INTERFACE itfAxis_Tc2_MC2

METHOD AbortTrigger : itfCommand
VAR_INPUT
END_VAR
END_METHOD

{attribute 'TcRpcEnable'}
METHOD AccelerationProfile 	: itfCommand
VAR_INPUT
	TimeScale				: REAL;
	AccelerationScale		: REAL;
	Offset					: REAL;
	BufferMode				: MC_BUFFER_MODE;
END_VAR
END_METHOD

{warning 'add property implementation'}
PROPERTY ActualPosition : REAL
GET
END_GET
END_PROPERTY

{warning 'add property implementation'}
PROPERTY ActualTorque : REAL
GET
END_GET
END_PROPERTY

{warning 'add property implementation'}
PROPERTY ActualVelocity : REAL
GET
END_GET
END_PROPERTY

{warning 'add property implementation'}
PROPERTY AxisWarning : BOOL
GET
END_GET
END_PROPERTY

{attribute 'TcRpcEnable'}
METHOD CombineAxes 			: itfSynchronizedAxisCommand
VAR_INPUT
	Master1					: itfAxis_Tc2_MC2;
	Master2					: itfAxis_Tc2_MC2;
	CombineMode				: MC_COMBINE_MODE;
	GearRatioNumeratorM1	: INT;
	GearRatioDenominatorM1	: INT;
	GearRatioNumeratorM2	: INT;
	GearRatioDenominatorM2	: INT;
	MasterValueSourceM1		: MC_SOURCE;
	MasterValueSourceM2		: MC_SOURCE;
	BufferMode				: MC_BUFFER_MODE;
END_VAR
END_METHOD

{warning 'add property implementation'}
PROPERTY CommunicationReady : BOOL
GET
END_GET
END_PROPERTY

{warning 'add property implementation'}
PROPERTY Direction : AXIS_DIRECTION
GET
END_GET
END_PROPERTY

PROPERTY Error : BOOL
GET
END_GET
END_PROPERTY

{warning 'add property implementation'}
PROPERTY ErrorId : WORD
GET
END_GET
END_PROPERTY

PROPERTY ErrorId_Udint_Status : UDINT
GET
END_GET
END_PROPERTY

PROPERTY Geared : BOOL
GET
END_GET
END_PROPERTY

{attribute 'TcRpcEnable'}
METHOD GearIn 			: itfSynchronizedAxisCommand
VAR_INPUT
//	Master				: itfAxis;
//	Master				: Tc2_MC2.AXIS_REF;
//	Slave				: Tc2_MC2.AXIS_REF;		
//	Ratio				: REAL;
//	MasterValueSource	: INT;
	RatioNumerator		: LREAL;
	RatioDenominator	: UINT;
	Acceleration		: REAL;
	Deceleration		: REAL;
	Jerk				: REAL;
	BufferMode			: MC_BUFFER_MODE;
//	BufferMode			: Tc2_MC2.MC_BufferMode;
//	Options             : Tc2_MC2.ST_GearInOptions;
END_VAR

VAR_IN_OUT 
	Slave				: Tc2_MC2.AXIS_REF;	
END_VAR
END_METHOD

{attribute 'TcRpcEnable'}
METHOD Halt 		: itfAxisCommand
VAR_INPUT
	Deceleration	: REAL;
	Jerk			: REAL;
	BufferMode		: MC_BUFFER_MODE;
END_VAR
END_METHOD

{attribute 'TcRpcEnable'}
METHOD HaltSuperimposed : itfAxisCommand
VAR_INPUT
	Deceleration		: REAL;
	Jerk				: REAL;
END_VAR
END_METHOD

{attribute 'TcRpcEnable'}
METHOD Home 		: itfAxisCommand
VAR_INPUT
	Position		: REAL;
	Velocity		: REAL;
	EndVelocity		: REAL;
	Acceleration	: REAL;
	Deceleration	: REAL;
	Jerk			: REAL;
	Direction		: MC_Direction;
	HomingMode		: INT;
	BufferMode		: MC_BUFFER_MODE;
END_VAR
END_METHOD

{warning 'add property implementation'}
PROPERTY HomeAbsSwitch : BOOL
GET
END_GET
END_PROPERTY


PROPERTY IsHomed : BOOL
GET
END_GET
END_PROPERTY

{attribute 'TcRpcEnable'}
METHOD Jog 			: itfAxisCommand
VAR_INPUT
    JogForward 		: BOOL;
    JogBackwards 	: BOOL;
    Mode     		: Tc2_MC2.E_JogMode;
    Position        : LREAL;
    Velocity        : LREAL;
    Acceleration 	: LREAL;
    Deceleration 	: LREAL;
    Jerk     		: LREAL;
END_VAR
END_METHOD

{warning 'add property implementation'}
PROPERTY LimitSwitchNegative : BOOL
GET
END_GET
END_PROPERTY

{warning 'add property implementation'}
PROPERTY LimitSwitchPositive : BOOL
GET
END_GET
END_PROPERTY

{warning 'add property implementation'}
PROPERTY MotionStatus : MOTION_STATUS
GET
END_GET
END_PROPERTY

{attribute 'TcRpcEnable'}
METHOD MoveAbsolute : itfAxisCommand
//METHOD ABSTRACT MoveAbsolute : itfAxisCommand
VAR_INPUT
	Position		: REAL;
	Velocity		: REAL;
	Acceleration	: REAL;
	Deceleration	: REAL;
	Jerk			: REAL;
//	Direction		: MC_Direction;
	BufferMode		: MC_BUFFER_MODE;
	Options         : Tc2_MC2.ST_MoveOptions;
END_VAR
END_METHOD

{attribute 'TcRpcEnable'}
METHOD MoveAdditive : itfAxisCommand
VAR_INPUT
	Distance		: REAL;
	Velocity		: REAL;
	Acceleration	: REAL;
	Deceleration	: REAL;
	Jerk			: REAL;
	BufferMode		: MC_BUFFER_MODE;
END_VAR
END_METHOD

{attribute 'TcRpcEnable'}
METHOD MoveContinuousAbsolute 	: itfContinuousAxisCommand
VAR_INPUT
	Position					: REAL;
	EndVelocity					: REAL;
	Velocity					: REAL;
	Acceleration				: REAL;
	Deceleration				: REAL;
	Jerk						: REAL;
	Direction					: MC_DIRECTION;
	BufferMode					: MC_BUFFER_MODE;
END_VAR
END_METHOD

{attribute 'TcRpcEnable'}
METHOD MoveContinuousRelative 	: itfContinuousAxisCommand
VAR_INPUT
	Distance					: REAL;
	EndVelocity					: REAL;
	Velocity					: REAL;
	Acceleration				: REAL;
	Deceleration				: REAL;
	Jerk						: REAL;
	Direction					: MC_DIRECTION;
	BufferMode					: MC_BUFFER_MODE;
END_VAR
END_METHOD

{attribute 'TcRpcEnable'}
METHOD MoveModulo : itfAxisCommand
VAR_INPUT
END_VAR
END_METHOD

{attribute 'TcRpcEnable'}
METHOD MoveRelative : itfAxisCommand
VAR_INPUT
	Distance		: REAL;
	Velocity		: REAL;
	Acceleration	: REAL;
	Deceleration	: REAL;
	Jerk			: REAL;
	BufferMode		: MC_BUFFER_MODE;
	Options         : Tc2_MC2.ST_MoveOptions;
END_VAR
END_METHOD

{attribute 'TcRpcEnable'}
METHOD MoveSuperimposed : itfAxisCommand
VAR_INPUT
	Distance			: REAL;
	VelocityDiff		: REAL;
	Acceleration		: REAL;
	Deceleration		: REAL;
	Jerk				: REAL;
END_VAR
END_METHOD

{attribute 'TcRpcEnable'}
METHOD MoveVelocity : itfContinuousAxisCommand
VAR_INPUT
	Velocity		: REAL;
	Acceleration	: REAL;
	Deceleration	: REAL;
	Jerk			: REAL;
	Direction		: MC_Direction;
	BufferMode		: MC_BUFFER_MODE;
END_VAR
END_METHOD

{attribute 'TcRpcEnable'}
METHOD PhasingAbsolute 	: itfSynchronizedAxisCommand
VAR_INPUT
//	Master				: itfAxis;
	Master				: Tc2_MC2.AXIS_REF;
	Slave				: Tc2_MC2.AXIS_REF;		
	PhaseShift			: REAL;
	Velocity			: REAL;
	Acceleration		: REAL;
	Deceleration		: REAL;
	Jerk				: REAL;
	BufferMode			: MC_BUFFER_MODE;
END_VAR
END_METHOD

{attribute 'TcRpcEnable'}
METHOD PhasingRelative 	: itfSynchronizedAxisCommand
VAR_INPUT
//	Master				: itfAxis;
	Master				: Tc2_MC2.AXIS_REF;
	Slave				: Tc2_MC2.AXIS_REF;		
	PhaseShift			: REAL;
	Velocity			: REAL;
	Acceleration		: REAL;
	Deceleration		: REAL;
	Jerk				: REAL;
	BufferMode			: MC_BUFFER_MODE;
END_VAR
END_METHOD

{attribute 'TcRpcEnable'}
METHOD PositionProfile : itfCommand
VAR_INPUT
	TimeScale			: REAL;
	PositionScale		: REAL;
	Offset				: REAL;
	BufferMode			: MC_BUFFER_MODE;
END_VAR
END_METHOD

{attribute 'TcRpcEnable'}
//METHOD ABSTRACT Power	: itfCommand
METHOD Power	: itfCommand
VAR_INPUT
	Enable				: BOOL;
	EnablePositive		: BOOL;
	EnableNegative		: BOOL;
END_VAR
END_METHOD

{attribute ‘monitoring’ := ‘call’}
PROPERTY PowerOn : BOOL
GET
END_GET
END_PROPERTY

{attribute 'TcRpcEnable'}
METHOD ReadBoolParameter 	: MC_Error
VAR_INPUT
	ParameterNumber			: INT;
END_VAR
VAR_OUTPUT
	Value					: BOOL;
END_VAR
END_METHOD

{attribute 'TcRpcEnable'}
METHOD ReadParameter 	: MC_Error
VAR_INPUT
	ParameterNumber		: INT;
END_VAR
VAR_OUTPUT
	Value				: REAL;
END_VAR
END_METHOD

{warning 'add property implementation'}
PROPERTY ReadyForPowerOn : BOOL
GET
END_GET
END_PROPERTY

{attribute 'TcRpcEnable'}
METHOD Release : MC_Error
END_METHOD

{attribute 'TcRpcEnable'}
METHOD Reset : itfCommand
END_METHOD

{attribute 'TcRpcEnable'}
METHOD SetOverride 	: MC_Error
VAR_INPUT
	VelFactor		: REAL;
	AccFactor		: REAL;
	JerkFactor		: REAL;
END_VAR
END_METHOD

{attribute 'TcRpcEnable'}
METHOD SetPosition 	: itfCommand
VAR_INPUT
	Position		: REAL;
	Relative		: BOOL;
//	ExecutionMode	: MC_ExecutionMode;
	ExecutionMode	: Tc2_MC2.ST_SetPositionOptions;
END_VAR
END_METHOD

{warning 'add property implementation'}
PROPERTY Simulation : BOOL
GET
END_GET
END_PROPERTY

PROPERTY Status : MC_AxisStates
GET
END_GET
END_PROPERTY

{attribute 'TcRpcEnable'}
METHOD Stop 		: itfAxisCommand
VAR_INPUT
	Deceleration	: REAL;
	Jerk			: REAL;
END_VAR
END_METHOD

{attribute 'TcRpcEnable'}
METHOD TorqueControl	: itfAxisCommand
VAR_INPUT
	Torque				: REAL;
	TorqueRamp			: REAL;
	Velocity			: REAL;
	Acceleration		: REAL;
	Deceleration		: REAL;
	Jerk				: REAL;
	Direction			: MC_DIRECTION;
	BufferMode			: MC_BUFFER_MODE;
END_VAR
END_METHOD

METHOD TouchProbe : itfCommand
VAR_INPUT
END_VAR
END_METHOD

{attribute 'TcRpcEnable'}
METHOD VelocityProfile 	: itfCommand
VAR_INPUT
	TimeScale			: REAL;
	VelocityScale		: REAL;
	Offset				: REAL;
	BufferMode			: MC_BUFFER_MODE;
END_VAR
END_METHOD

{attribute 'TcRpcEnable'}
METHOD WriteBoolParameter 	: MC_Error
VAR_INPUT
	ParameterNumber			: INT;
	Value					: BOOL;
END_VAR
END_METHOD

{attribute 'TcRpcEnable'}
METHOD WriteParameter 	: MC_Error
VAR_INPUT
	ParameterNumber		: INT;
	Value				: REAL;
END_VAR
END_METHOD

END_INTERFACE

(* stored: Version 1.1.0.1, ProductVersion 3.1.4024.12
   Itf itfAxis_Tc2_MC2: Id {61cb14c2-e05e-4264-a99b-c2e5bed78828}
   Folder ActualValues: Id {12d21fd6-9367-490a-a5c0-f3d812c9e60d}
   Folder Control: Id {7f975a5b-2041-480a-8274-c87ae9d6cf4c}
   Folder MultiAxesMotion: Id {c3a2a744-de13-424f-9539-31f81d1d61b6}
   Folder SingleAxisMotion: Id {abafcda8-9d6d-45cf-afd2-2c702b3f6ac0}
   Folder Status: Id {023fc74a-643f-4641-afcf-b66559b00ebc}
   Folder Touch Probe: Id {88a0a759-a042-40a5-9f66-3353ee0d1693}
   Method AbortTrigger: Id {39b56d76-08fa-4a19-bfca-878a60803512}
   Method AccelerationProfile: Id {df31f7b2-0556-40dc-b14a-854531e29ed5}
   Property ActualPosition: Id {d13ea898-23c4-443f-ae50-f01fe1b2508c}
   Get Get: Id {48219e97-9494-4bd8-9c8b-ded0f45ec504}
   Property ActualTorque: Id {2b661e49-afcc-491e-b1c7-0c13296e7c90}
   Get Get: Id {cb0b144c-5ef5-4c4d-be6c-23304724dfd8}
   Property ActualVelocity: Id {1fef0271-409c-4e96-8705-62cc913eff3d}
   Get Get: Id {4b1aae3a-b02c-4d34-9a5e-995806437b3a}
   Property AxisWarning: Id {d1a1ba79-e96a-425b-a654-e329ba26c187}
   Get Get: Id {4b31a212-2efc-4626-b24d-837a9f312305}
   Method CombineAxes: Id {c33a9fa2-effc-4321-ac46-ce9c88fb47c7}
   Property CommunicationReady: Id {db527b3d-8967-4407-9224-84b327558cc1}
   Get Get: Id {00ca901e-d6bb-47d0-bd66-e6d2d82c2aca}
   Property Direction: Id {3b6184b0-6440-413c-9e0a-5d299ca03442}
   Get Get: Id {0df2cdbc-db86-447b-8a76-e8ca7704c856}
   Property Error: Id {5c8d6528-5ce4-4473-884d-43d29fb7b151}
   Get Get: Id {9dbcafe8-ae1e-400f-b0c2-40e38822dafc}
   Property ErrorId: Id {f3c50114-fdd3-4d45-8328-ccd9b9533a9e}
   Get Get: Id {937c6632-549c-4a5c-9cc4-9fc45cb9d853}
   Property ErrorId_Udint_Status: Id {3526cd07-fc61-423c-ae5b-33630528fd91}
   Get Get: Id {5472ad64-8f30-439c-a73c-1cf30cb6d6e6}
   Property Geared: Id {c8ab79e2-22f2-4c0b-ab80-2b08fcd8d983}
   Get Get: Id {23cf5cc3-0a54-486a-9302-6865f9e9426d}
   Method GearIn: Id {c95c1128-9524-4448-a3ec-30a5218a30e7}
   Method Halt: Id {42e9015f-9078-4397-a6ff-f6f6026ddfea}
   Method HaltSuperimposed: Id {d68cb379-a128-40e2-beca-7c4e6ddd88e0}
   Method Home: Id {7d680615-a29d-494e-aeca-d386a520986c}
   Property HomeAbsSwitch: Id {01475c57-20c5-4952-841c-1bc14f17fae3}
   Get Get: Id {ba267200-ec64-41f0-89b7-63529568456f}
   Property IsHomed: Id {f4be05eb-d7e8-4d42-ab4a-d900b029e078}
   Get Get: Id {b5c49bd4-9690-48a2-a915-526f757ee4e6}
   Method Jog: Id {69f9cbd4-3391-4431-b95f-62e9da8ec880}
   Property LimitSwitchNegative: Id {17b135cf-f40c-47bc-99fe-7894888dd695}
   Get Get: Id {d83785f0-59d3-4802-82fc-bdef3951b18a}
   Property LimitSwitchPositive: Id {0478b642-44c4-4560-a8d1-9d0e046a9fe2}
   Get Get: Id {04afa5cd-b1cb-4d45-959a-f5a3620cd165}
   Property MotionStatus: Id {dad19ba9-c17e-449a-b44a-638d4ee2b270}
   Get Get: Id {9ebac635-8754-450e-803b-159110d87cea}
   Method MoveAbsolute: Id {603952a0-b0c9-4314-be40-2176144ec08d}
   Method MoveAdditive: Id {82801e35-f9f5-4d17-9c52-2ad8fb992b71}
   Method MoveContinuousAbsolute: Id {cab2631a-6b16-4d7b-97d2-b3ef1a50638a}
   Method MoveContinuousRelative: Id {e243a40a-6895-4c97-9537-990d7389ad60}
   Method MoveModulo: Id {98915bb3-c786-4bca-922a-8e77ba1376a8}
   Method MoveRelative: Id {32213576-2ddc-491e-b2d3-e2ba8f82726a}
   Method MoveSuperimposed: Id {e6ebe6d8-b482-4321-acf9-4b22df4a9581}
   Method MoveVelocity: Id {0a80f606-6a8b-4fe2-bae8-d2e83e641674}
   Method PhasingAbsolute: Id {83de4694-0ed4-470c-8084-9521fb186863}
   Method PhasingRelative: Id {f386ddd5-736e-4e7c-8a62-1e5046c596d3}
   Method PositionProfile: Id {19b92d91-811d-4e6f-9bbf-f46faa803b76}
   Method Power: Id {75fd3267-1b9f-4a40-a69d-fe4a6a848e6c}
   Property PowerOn: Id {3d0df34b-1501-472d-a293-28a40bc36f88}
   Get Get: Id {ca190771-b66c-4413-916b-44392df4187c}
   Method ReadBoolParameter: Id {13dfcb7a-9fca-42a9-9019-a3f4052bfe8c}
   Method ReadParameter: Id {c5b548c4-a9c4-44cb-b222-a03f23b47bcb}
   Property ReadyForPowerOn: Id {e29db299-083f-413f-a629-2bb7708d005f}
   Get Get: Id {1cfbfd59-e9df-44a9-b69e-b4d7ed1cacd5}
   Method Release: Id {50052424-1f88-4c87-b31a-991d95e0a89f}
   Method Reset: Id {e890dd0a-f2c8-4af3-b70c-e29a653734d4}
   Method SetOverride: Id {1c09732f-7e62-4d8f-b8f9-e500a69291f3}
   Method SetPosition: Id {d7c0c6ee-111f-412f-81b8-ec5a0a44f6fb}
   Property Simulation: Id {f2d687fb-12c1-4b4f-b6ac-e8d2a28e5370}
   Get Get: Id {a077cdc3-47a9-44b4-a459-909c1f30918e}
   Property Status: Id {c79a357d-48d3-46f6-b508-c92730160c3c}
   Get Get: Id {c4cfb2af-4adb-43b4-9726-207a1f048f4e}
   Method Stop: Id {075b8b04-d3dd-4136-9cf7-793879b8df29}
   Method TorqueControl: Id {e40b1b18-f414-42ef-ad98-67224ac9a31a}
   Method TouchProbe: Id {9dce40a0-7b6e-42d5-8801-1abf14002266}
   Method VelocityProfile: Id {e9f3e391-a484-4147-82be-c9fb21ffd36a}
   Method WriteBoolParameter: Id {e455080b-9cbe-445c-98e5-c78faebf683b}
   Method WriteParameter: Id {97fcd37b-6856-4802-a866-95a897e19fed} *)
